TYPE AxesConfigs :
STRUCT
	IoStageAxisConfig : IoStageAxisConfig;	
	Ps10OwisAxisConfig : Ps10OwisAxisConfig;
END_STRUCT
END_TYPE

(* stored: Version 1.1.0.1, ProductVersion 3.1.4024.12
   DUT AxesConfigs: Id {b89ab97d-6cd8-4401-a62d-09f9a0d5372c} *)
